SUBAPPLICATION Uebung_039b (* Spiegelabfolge V2 mit Schrittkette *)
  (* Standard: 61499-2; Description: Spiegelabfolge V2 mit Schrittkette geeignet für hydraulisches Ringsystem 3/2 Wege Ventile  (z.B. Claas) oder pneumatische 5/2 Wege Ventile *)
  (* Version 1.0, 2023-10-23, franz *)
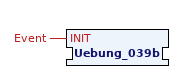
  EVENT_INPUT
    INIT;
  END_EVENT
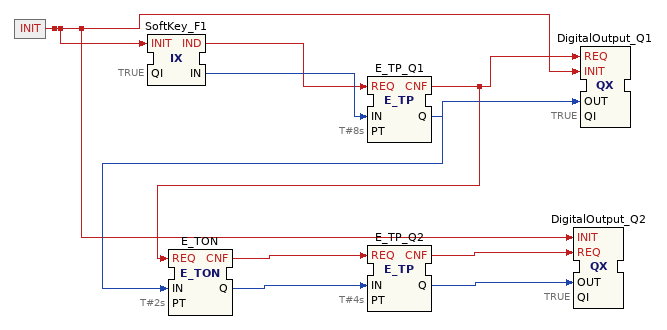
  FBS
    DigitalOutput_Q1 : QX(QI := TRUE);
    DigitalOutput_Q2 : QX(QI := TRUE);
    SoftKey_F1 : IX(QI := TRUE);
    E_TP_Q1 : E_TP(PT := T#8s);
    E_TP_Q2 : E_TP(PT := T#4s);
    E_TON : E_TON(PT := T#2s);
  END_FBS
  EVENT_CONNECTIONS
    INIT TO SoftKey_F1.INIT;
    E_TP_Q1.CNF TO DigitalOutput_Q1.REQ;
    INIT TO DigitalOutput_Q1.INIT;
    INIT TO DigitalOutput_Q2.INIT;
    E_TP_Q2.CNF TO DigitalOutput_Q2.REQ;
    E_TP_Q1.CNF TO E_TON.REQ;
    E_TON.CNF TO E_TP_Q2.REQ;
    SoftKey_F1.IND TO E_TP_Q1.REQ;
  END_CONNECTIONS
  DATA_CONNECTIONS
    E_TP_Q2.Q TO DigitalOutput_Q2.OUT;
    E_TP_Q1.Q TO DigitalOutput_Q1.OUT;
    E_TP_Q1.Q TO E_TON.IN;
    E_TON.Q TO E_TP_Q2.IN;
    SoftKey_F1.IN TO E_TP_Q1.IN;
  END_CONNECTIONS
END_SUBAPPLICATION
